INTERFACE I_PositionalDrive EXTENDS I_Drive

PROPERTY CurrentPosition : LREAL
GET
END_GET
END_PROPERTY

METHOD ABSTRACT moveAbsolute : BOOL
VAR_INPUT
	newTarget : LREAL; 
END_VAR
END_METHOD

METHOD ABSTRACT moveRelative : BOOL
VAR_INPUT
	distance : LREAL;
END_VAR
END_METHOD

METHOD setPosition : BOOL
VAR_INPUT
	newPosition : LREAL;
END_VAR
END_METHOD

PROPERTY TargetPosition : LREAL
GET
END_GET
END_PROPERTY

END_INTERFACE

(* stored: Version 1.1.0.1, ProductVersion 3.1.4024.11
   Itf I_PositionalDrive: Id {81a09306-99e6-4c4b-9cae-7e4ea95c241a}
   Folder Properties: Id {de147b7a-07e6-4251-88fb-4cfe388e42ae}
   Property CurrentPosition: Id {f078ea92-8635-4370-a27c-8f25163069aa}
   Get Get: Id {e3426102-b935-427b-9621-f0ea6e15d792}
   Method moveAbsolute: Id {9a9cdf6d-aec6-44ca-984d-f7b16f0af7b8}
   Method moveRelative: Id {981b39f0-30e4-4cef-ab4a-d99e9e3c1753}
   Method setPosition: Id {a624681b-c3ac-4d17-9436-29c905c19776}
   Property TargetPosition: Id {83da7a30-d7ab-4526-8c71-3fc27340b980}
   Get Get: Id {23036b62-7b0c-4685-a416-054cbcc4179e} *)
